TYPE ST_TwoHandParCmd :
STRUCT
    Reserved : BOOL;
END_STRUCT
END_TYPE

(* stored: Version 1.1.0.1, ProductVersion 3.1.4024.12
   DUT ST_TwoHandParCmd: Id {88c519d2-f2e9-44c0-9ab0-169ec26d2464} *)
